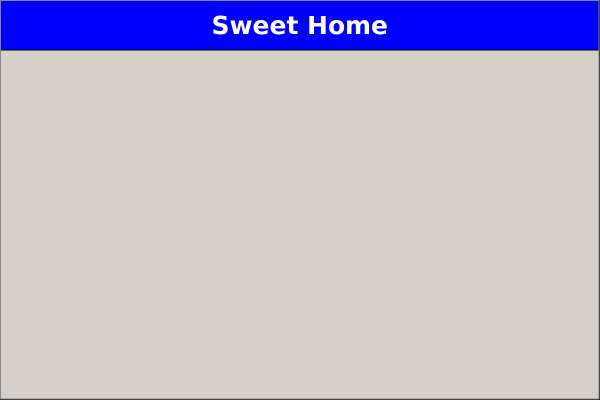
VISUALIZATION Template  // 600x400
    Rectangle (0,0 600x400)
    Rectangle (0,0 600x50), "Sweet Home"
END_VISUALIZATION

(* stored: Version 1.1.0.1, ProductVersion 3.1.4024.12
   Visu Template: Id {270002af-43d2-42b2-9705-3df7410e3517} *)
